{attribute 'GeneratedUsingTerminal: EP1816-0003-0016'}
{attribute addProperty BoxType "EP1816-0003-0016"}
{attribute addProperty Id "DIG_Inputs_Channel_1AT %I*DIG_Inputs_Channel_ACAA042510DIG_Inputs_Channel_2AT %I*DIG_Inputs_Channel_ACAA042510WcStateAT %I*WcState_9091E0EB2InfoDataAT %I*InfoData_94A18F5E2"}
{attribute addProperty CRC "2492605939"}
{attribute addProperty Size "24"}
TYPE EP1816_949225F3 EXTENDS EtcSlaveTerminalBase_947E5A46 :
STRUCT
	{attribute addProperty Name "DIG_Inputs_Channel_1"}
	DIG_Inputs_Channel_1 : DIG_Inputs_Channel_ACAA0425;
	{attribute addProperty Name "DIG_Inputs_Channel_2"}
	DIG_Inputs_Channel_2 : DIG_Inputs_Channel_ACAA0425;
	{attribute addProperty Name "WcState"}
	WcState : WcState_9091E0EB;
	{attribute addProperty Name "InfoData"}
	InfoData : InfoData_94A18F5E;
END_STRUCT
END_TYPE

(* stored: Version 1.2.0.0, ProductVersion 3.1.4024.9
   DUT EP1816_949225F3: Id {3968b85b-83c8-42eb-95e9-72b10d292ad9} *)
